FUNCTION_BLOCK FB_GcodeAgent
VAR_INPUT
	bExecute : BOOL;
	bNextLine : BOOL;
	bWriteDone : BOOL;
	sGcodeFile : STRING;
	sFBName : STRING;
	bEnd : BOOL;
END_VAR
VAR_OUTPUT
	x : REAL;
	y : REAL;
	z : REAL;
	e : REAL;
	f : REAL;
END_VAR
VAR
	trig : R_TRIG;
	Process : NT_StartProcess;
	sCommand : STRING(1000);
	placeholder : ARRAY [0..200] OF STRING(200);
END_VAR
//'main.py choppt.gcode MovementTypeSelector.fbGcode.gcodeagent 10.123.67.6.1.1'

// prepare command to run python script]
trig(CLK := bExecute);
placeholder[0] := sGcodeFile;
placeholder[1] := ' ';
placeholder[2] := sFBName;
placeholder[3] := ' ';
placeholder[4] := HbotForwardKinematics.fbAms.AddrString;

sCommand := ConcatAll(placeholder); //concat all

Process(NETID := '10.123.6.66.1.1',
		COMNDLINE := sCommand,
		PATHSTR := 'C:\Users\weikoons.BECKHOFF\Downloads\HBot_SelfDefinedKinematics\HBot_SelfDefinedKinematics\Hboy\POUs\MovementType_Gcode\main.exe',
//		DIRNAME := 'C:\Users\MaxwellA.BECKHOFF\Desktop\Coding\Python\asd\Gcode',
		START := trig.Q); // start process

METHOD ConcatAll : STRING(1000)
VAR_INPUT
	allString : ARRAY [0..200] OF STRING(200);
END_VAR
VAR
	resultString : STRING(1000);
	i : INT;
END_VAR
FOR i := 0 TO 199 DO
	IF allString[i] = '' THEN
		ConcatAll := resultString;
	END_IF
	resultString := CONCAT(resultString, allString[i]);
END_FOR
ConcatAll := resultString;
END_METHOD

END_FUNCTION_BLOCK

(* stored: Version 1.1.0.1, ProductVersion 3.1.4024.11
   POU FB_GcodeAgent: Id {76f8f1b8-8bc2-46fa-945f-c481147d0a02}, SpecialFunc None
   Method ConcatAll: Id {745a41d0-fcb4-41c1-b418-a68acb14b841} *)
